FUNCTION F_ITC_SendSNR : BOOL
(**************************************************************************************
 * 	Application		:	BoxControl Framework
 *	Revision		:	$Revision: 404529 $
 *	Revision date	:	$Date: 2018-04-23 08:21:38 +0200 (Mo., 23 Apr 2018) $
 *	Last changed by	:	$Author: b7bolm $
 *	URL				:	$URL: http://almscdc.swisslog.com/repo/SWPD/Development/BoxControlFramework/20_Release/trunk/01_Software/BCF/BCF/JumpStart/20_Product/10_App/11_Com/10_Lib/10_Conv/11_ITC/F_ITC_SendSNR.TcPOU $
 *
 *	Purpose			:	Wrap message - SNR
 *
 * ------------------------------------------------------------------------------------
 *	Copyright Swisslog [IP AG], Switzerland. All rights reserved.
 * 
 * ------------------------------------------------------------------------------------
 *	
 * 	Revision History: 
 *
 * 	VERSION			DATE			INITIALS			DESCRIPTION
 *	0.1				01.01.2001		swl					Example
 *
 **************************************************************************************)
VAR_INPUT
	eChannelSrc		: E_MFCS_Channel; // Source communicaton channel	
	PositionName	: STRING(Conveyor.POSITION_STRINGLENGTH); // Position
	TU_ID			: STRING(Conveyor.TU_ID_STRINGLENGTH); // TU ID
	eInfoCode		: E_ErrorConv; // Info Code
END_VAR
VAR
	SNR				: ST_ITC_SNR; 
END_VAR

// Map values
SNR.Position := PositionName;
SNR.TU_ID := TU_ID;
SNR.InfoCode := eInfoCode;

// Forward to ITC
F_ITC_SendSNR := fbITC_Manager.M_SendData(
					meChannel	:= eChannelSrc,
					mMsgType	:= E_ITC_MsgTypeConv.SCANNER_NO_READ_REPORT,
					mpData		:= ADR(SNR),
					mLen		:= SIZEOF(SNR));

END_FUNCTION

(* stored: Version 1.1.0.1, ProductVersion 3.1.4022.12
   POU F_ITC_SendSNR: Id {12a9420f-0328-43a1-9ddc-4e217729f4c6}, SpecialFunc None *)
